TYPE tyRampInputs :
STRUCT
	bActivateRamp : BOOL; 
	bResetRamp :BOOL; 
	iNumberOfSteps : INT ;
	tRampProgramTimeLimit : time ;
END_STRUCT
END_TYPE

(* stored: Version 1.1.0.1
   DUT tyRampInputs: Id {c43b9272-8d53-4178-8184-24b69009a6f0} *)
